Staubli VAL3: searchL.pgx

public program searchL(point x_pEndSearch, tool x_tTool, mdesc x_mMdesc, frame& x_fFrame, dio x_dInput, point& x_pFound)
  local mdesc l_mMdesc
begin

  //execute a movel from x_pStartSearch to x_pEndSearch
  //if x_dInput switch to true during this movement the robot stops and the current position of x_tTool is written in x_pFound
  //note: x_dInput isn't necessarily an input, the blend of the movement is set to off by default

  bSearchLFail=false
  bSearchLSuccess=false

  if taskStatus("searchL")==-1
    taskCreate "searchL",10,exeSearchL(x_dInput,x_tTool)
  else
    logMsg("libSignals/searchL->error creating the control task")
  endIf

  l_mMdesc=x_mMdesc
  l_mMdesc.blend=off

  movel(x_pEndSearch,x_tTool,l_mMdesc)
  wait(distance(here(x_tTool,x_fFrame),x_pEndSearch)<nBlendOffToll or bSearchLSuccess)
  if !bSearchLSuccess
    bSearchLFail=true
  else
    x_pFound=here(x_tTool,x_fFrame)
  endIf
end
